TYPE ST_BladePositionsEncoder :
STRUCT
bExtremeFeather_Exceeded	:BOOL;		
bExtremeFeather		:BOOL;
bFeather		:BOOL;
bExtremeFine	:BOOL;
bExtremeFine_Exceeded	:BOOL;

END_STRUCT
END_TYPE

(* stored: Version 1.1.0.1, ProductVersion 3.1.4024.9
   DUT ST_BladePositionsEncoder: Id {ddb12c86-b8dd-4ed3-99c1-095d290486de} *)
